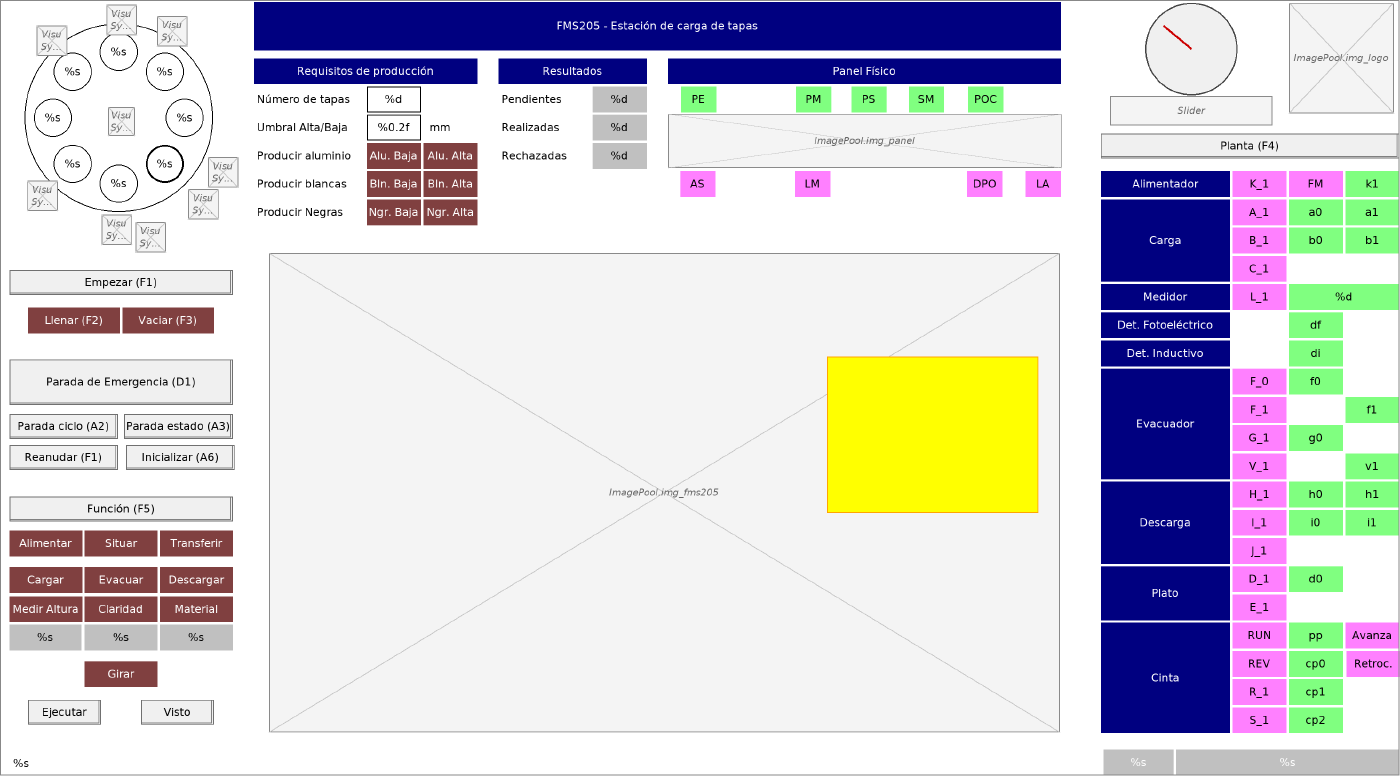
VISUALIZATION fms205visu  // 1488x825
    Rectangle (270,2 857x51), "FMS205 - Estación de carga de tapas", colour variable: MAIN.fbFMS205.dr.gmModeColor
        p3450524324: MAIN.fbFMS205.dr.gmModeColor
    Rectangle (270,62 237x27), "Requisitos de producción"
    Rectangle (530,62 157x27), "Resultados"
    Rectangle (710,62 417x27), "Panel Físico"
    Rectangle (270,92 157x27), "Número de tapas"
    Rectangle (390,92 57x27), "%d", text variable: MAIN.fbFMS205.ProdRequerida
    Rectangle (530,92 97x27), "Pendientes"
    Rectangle (630,92 57x27), "%d", text variable: MAIN.fbFMS205.ProdPendiente
    Rectangle (724,92 37x27), "PE", input disabled if: NOT MAIN.fbFMS205.dr.gmLocalHost
        toggle MAIN.fbFMS205.fbPanel.hwPE_Seta
    Rectangle (1029,92 37x27), "POC", input disabled if: NOT MAIN.fbFMS205.dr.gmLocalHost
        toggle MAIN.fbFMS205.fbPanel.hw.POC_PulsadorReset
    Rectangle (846,92 37x27), "PM", input disabled if: NOT MAIN.fbFMS205.dr.gmLocalHost
        toggle MAIN.fbFMS205.fbPanel.hw.PM_PulsadorMarcha
    Rectangle (966,92 37x27), "SM", input disabled if: NOT MAIN.fbFMS205.dr.gmLocalHost
        toggle MAIN.fbFMS205.fbPanel.hw.SM_SelecAutoManual
    Rectangle (270,122 117x27), "Umbral Alta/Baja"
    Rectangle (390,122 57x27), "%0.2f", text variable: MAIN.fbFMS205.fbPanel.cnUmbralAlta
        p4168582468: 'Atura en mm mínima para considerar que la tapa es alta'
    Rectangle (450,122 37x27), "mm"
    Rectangle (530,122 117x27), "Realizadas"
    Rectangle (630,122 57x27), "%d", text variable: MAIN.fbFMS205.ProdRealizada
    Rectangle (270,152 117x27), "Producir aluminio"
    Rectangle (390,152 57x27), "Alu. Baja"
        toggle MAIN.fbFMS205.fbPanel.cnProdAluBaja
    Rectangle (450,152 57x27), "Alu. Alta"
        toggle MAIN.fbFMS205.fbPanel.cnProdAluAlta
    Rectangle (530,152 117x27), "Rechazadas"
    Rectangle (630,152 57x27), "%d", text variable: MAIN.fbFMS205.ProdRechazada
    Button (1170,142 317x26), "Planta (F4)", tooltip "%s"
        p4168582468: MAIN.fbFMS205.fbPanel.ttF4_Planta
        toggle MAIN.fbFMS205.fbPanel.swF4_Planta
    Rectangle (270,182 117x27), "Producir blancas"
    Rectangle (390,182 57x27), "Bln. Baja"
        toggle MAIN.fbFMS205.fbPanel.cnProdBlaBaja
    Rectangle (450,182 57x27), "Bln. Alta"
        toggle MAIN.fbFMS205.fbPanel.cnProdBlaAlta
    Rectangle (1170,182 137x27), "Alimentador"
    Rectangle (1310,182 57x27), "K_1", input disabled if: NOT MAIN.fbFMS205.fbPanel.cnF4_Planta
        toggle MAIN.fbFMS205.mdAlimentador.K_1.uiValue p2164770859=TRUE
    Rectangle (1370,182 57x27), "FM", input disabled if: NOT MAIN.fbFMS205.fbPanel.cnF4_Planta
        toggle MAIN.fbFMS205.mdAlimentador.FM.uiValue
    Rectangle (1430,182 57x27), "k1", input disabled if: NOT MAIN.fbFMS205.fbPanel.cnF4_Planta
        toggle MAIN.fbFMS205.mdAlimentador.k1.uiValue
    Rectangle (723,182 37x27), "AS", input disabled if: NOT MAIN.fbFMS205.dr.gmLocalHost
        toggle MAIN.fbFMS205.fbPanel.hw.AS_AvisadorSonoro
    Rectangle (845,182 37x27), "LM", input disabled if: NOT MAIN.fbFMS205.dr.gmLocalHost
        toggle MAIN.fbFMS205.fbPanel.hw.LM_LamparaMarcha
    Rectangle (1028,182 37x27), "DPO", input disabled if: NOT MAIN.fbFMS205.dr.gmLocalHost
        toggle MAIN.fbFMS205.mdMedidorTapa.L_1.uiValue
    Rectangle (1090,182 37x27), "LA", input disabled if: NOT MAIN.fbFMS205.dr.gmLocalHost
        toggle MAIN.fbFMS205.fbPanel.hw.LA_LamparaAlarma
    Rectangle (270,212 117x27), "Producir Negras"
    Rectangle (390,212 57x27), "Ngr. Baja"
        toggle MAIN.fbFMS205.fbPanel.cnProdNegBaja
    Rectangle (450,212 57x27), "Ngr. Alta"
        toggle MAIN.fbFMS205.fbPanel.cnProdNegAlta
    Rectangle (1170,212 137x87), "Carga"
    Rectangle (1310,212 57x27), "A_1", input disabled if: NOT MAIN.fbFMS205.fbPanel.cnF4_Planta
        toggle MAIN.fbFMS205.mdPickAndPlaceCarga.HOR.uiValue
    Rectangle (1370,212 57x27), "a0", input disabled if: NOT MAIN.fbFMS205.fbPanel.cnF4_Planta
        toggle MAIN.fbFMS205.mdPickAndPlaceCarga.h0.uiValue
    Rectangle (1430,212 57x27), "a1", input disabled if: NOT MAIN.fbFMS205.fbPanel.cnF4_Planta
        toggle MAIN.fbFMS205.mdPickAndPlaceCarga.h1.uiValue
    Rectangle (1310,242 57x27), "B_1", input disabled if: NOT MAIN.fbFMS205.fbPanel.cnF4_Planta
        toggle MAIN.fbFMS205.mdPickAndPlaceCarga.VER.uiValue
    Rectangle (1370,242 57x27), "b0", input disabled if: NOT MAIN.fbFMS205.fbPanel.cnF4_Planta
        toggle MAIN.fbFMS205.mdPickAndPlaceCarga.v0.uiValue
    Rectangle (1430,242 57x27), "b1", input disabled if: NOT MAIN.fbFMS205.fbPanel.cnF4_Planta
        toggle MAIN.fbFMS205.mdPickAndPlaceCarga.v1.uiValue
    Rectangle (286,269 837x507), "Estacion"
    Button (10,287 237x26), "Empezar (F1)"
    Rectangle (30,327 97x27), "Llenar (F2)"
        toggle MAIN.fbFMS205.dr.fun_Llenar
    Rectangle (130,327 97x27), "Vaciar (F3)"
        toggle MAIN.fbFMS205.dr.fun_Vaciar
    Button (10,382 237x48), "Parada de Emergencia (D1)", tooltip "%s"
        p4168582468: MAIN.fbFMS205.fbPanel.ttPE_Seta
        toggle MAIN.fbFMS205.fbPanel.swPE_Seta
    Button (10,440 115x26), "Parada ciclo (A2)", input disabled if: not MAIN.fbFMS205.fbPanel.enA2_FinCiclo
        toggle MAIN.fbFMS205.fbPanel.swA2_FinCiclo
    Button (132,440 115x26), "Parada estado (A3)", input disabled if: not MAIN.fbFMS205.fbPanel.enA3_Estado
        toggle MAIN.fbFMS205.fbPanel.swA3_Estado
    Rectangle (1310,272 57x27), "C_1", input disabled if: NOT MAIN.fbFMS205.dr.bot_Planta
        toggle MAIN.fbFMS205.mdPickAndPlaceCarga.PIN.uiValue
    Rectangle (1170,302 137x27), "Medidor"
    Rectangle (1310,302 57x27), "L_1", input disabled if: NOT MAIN.fbFMS205.fbPanel.cnF4_Planta
        toggle MAIN.fbFMS205.mdMedidorTapa.L_1.uiValue
    Rectangle (1370,302 117x27), "%d", text variable: MAIN.fbFMS205.mdMedidorTapa.dh, input disabled if: NOT MAIN.fbFMS205.fbPanel.cnF4_Planta
    Rectangle (1170,332 137x27), "Det. Fotoeléctrico"
    Rectangle (1370,332 57x27), "df", input disabled if: NOT MAIN.fbFMS205.fbPanel.cnF4_Planta
        toggle MAIN.fbFMS205.mdDetectorFotoelectrico.df.uiValue
    Rectangle (1170,362 137x27), "Det. Inductivo"
    Rectangle (1370,362 57x27), "di", input disabled if: NOT MAIN.fbFMS205.fbPanel.cnF4_Planta
        toggle MAIN.fbFMS205.mdCaptadorInductivo.di.uiValue
    Rectangle (1170,392 137x117), "Evacuador"
    Rectangle (1310,392 57x27), "F_0", input disabled if: NOT MAIN.fbFMS205.fbPanel.cnF4_Planta
        toggle MAIN.fbFMS205.mdEvacuador.F_0.uiValue
    Rectangle (1370,392 57x27), "f0", input disabled if: NOT MAIN.fbFMS205.fbPanel.cnF4_Planta
        toggle MAIN.fbFMS205.mdEvacuador.f0.uiValue
    Button (10,528 237x26), "Función (F5)"
        toggle MAIN.fbFMS205.fbPanel.swF5_Funcion
    Rectangle (1310,422 57x27), "F_1", input disabled if: NOT MAIN.fbFMS205.fbPanel.cnF4_Planta
        toggle MAIN.fbFMS205.mdEvacuador.F_1.uiValue
    Rectangle (1430,422 57x27), "f1", input disabled if: NOT MAIN.fbFMS205.fbPanel.cnF4_Planta
        toggle MAIN.fbFMS205.mdEvacuador.f1.uiValue
    Rectangle (10,564 77x27), "Alimentar", input disabled if: not MAIN.fbFMS205.fbPanel.cnF5_Funcion
        toggle MAIN.fbFMS205.fbPanel.swF5_Alimentar
    Rectangle (90,703 77x27), "Girar", input disabled if: not MAIN.fbFMS205.fbPanel.cnF5_Funcion
        toggle MAIN.fbFMS205.fbPanel.swF5_Girar
    Rectangle (90,564 77x27), "Situar", input disabled if: not MAIN.fbFMS205.fbPanel.cnF5_Funcion
        toggle MAIN.fbFMS205.fbPanel.swF5_Situar
    Rectangle (10,634 77x27), "Medir Altura", input disabled if: not MAIN.fbFMS205.fbPanel.cnF5_Funcion
        toggle MAIN.fbFMS205.fbPanel.swF5_Medir
    Rectangle (90,634 77x27), "Claridad", input disabled if: not MAIN.fbFMS205.fbPanel.cnF5_Funcion
        toggle MAIN.fbFMS205.fbPanel.swF5_Claridad
    Rectangle (170,634 77x27), "Material", input disabled if: not MAIN.fbFMS205.fbPanel.cnF5_Funcion
        toggle MAIN.fbFMS205.fbPanel.swF5_Material
    Rectangle (10,664 76x27), "%s", text variable: MAIN.fbFMS205.mdMedidorTapa.strUi
    Rectangle (90,664 77x27), "%s", text variable: MAIN.fbFMS205.mdDetectorFotoelectrico.strUi
    Rectangle (170,664 77x27), "%s", text variable: MAIN.fbFMS205.mdCaptadorInductivo.strUi
    Rectangle (10,603 77x27), "Cargar", input disabled if: not MAIN.fbFMS205.fbPanel.cnF5_Funcion
        toggle MAIN.fbFMS205.fbPanel.swF5_Cargar
    Rectangle (90,603 77x27), "Evacuar", input disabled if: not MAIN.fbFMS205.fbPanel.cnF5_Funcion
        toggle MAIN.fbFMS205.fbPanel.swF5_Evacuar
    Rectangle (170,603 77x27), "Descargar", input disabled if: not MAIN.fbFMS205.fbPanel.cnF5_Funcion
        toggle MAIN.fbFMS205.fbPanel.swF5_Descargar
    Rectangle (170,564 77x27), "Transferir", input disabled if: not MAIN.fbFMS205.fbPanel.cnF5_Funcion
        toggle MAIN.fbFMS205.fbPanel.swF5_Transferir
    Button (30,744 77x26), "Ejecutar", input disabled if: not MAIN.fbFMS205.fbPanel.cnF5_Funcion
        tap MAIN.fbFMS205.fbPanel.swF5_Ejecutar
    Button (150,744 77x26), "Visto", input disabled if: not MAIN.fbFMS205.fbPanel.cnF5_Funcion
        tap MAIN.fbFMS205.fbPanel.swF5_Ack
    Rectangle (1310,452 57x27), "G_1", input disabled if: NOT MAIN.fbFMS205.fbPanel.cnF4_Planta
        toggle MAIN.fbFMS205.mdEvacuador.G_1.uiValue
    Rectangle (1370,452 57x27), "g0", input disabled if: NOT MAIN.fbFMS205.fbPanel.cnF4_Planta
        toggle MAIN.fbFMS205.mdEvacuador.g0.uiValue
    Rectangle (1310,482 57x27), "V_1", input disabled if: NOT MAIN.fbFMS205.fbPanel.cnF4_Planta
        toggle MAIN.fbFMS205.mdEvacuador.V_1.uiValue
    Rectangle (1430,482 57x27), "v1", input disabled if: NOT MAIN.fbFMS205.fbPanel.cnF4_Planta
        toggle MAIN.fbFMS205.mdEvacuador.v1.uiValue
    Rectangle (1170,512 137x87), "Descarga"
    Rectangle (1310,512 57x27), "H_1", input disabled if: NOT MAIN.fbFMS205.fbPanel.cnF4_Planta
        toggle MAIN.fbFMS205.mdPickAndPlaceDescarga.HOR.uiValue
    Rectangle (1370,512 57x27), "h0", input disabled if: NOT MAIN.fbFMS205.fbPanel.cnF4_Planta
        tap MAIN.fbFMS205.mdPickAndPlaceDescarga.h0.uiValue
        toggle MAIN.fbFMS205.mdPickAndPlaceDescarga.h0.uiValue
    Rectangle (1430,512 57x27), "h1", input disabled if: NOT MAIN.fbFMS205.fbPanel.cnF4_Planta
        toggle MAIN.fbFMS205.mdPickAndPlaceDescarga.h1.uiValue
    Rectangle (1310,542 57x27), "I_1", input disabled if: NOT MAIN.fbFMS205.fbPanel.cnF4_Planta
        toggle MAIN.fbFMS205.mdPickAndPlaceDescarga.VER.uiValue
    Rectangle (1370,542 57x27), "i0", input disabled if: NOT MAIN.fbFMS205.fbPanel.cnF4_Planta
        toggle MAIN.fbFMS205.mdPickAndPlaceDescarga.v0.uiValue
    Rectangle (1430,542 57x27), "i1", input disabled if: NOT MAIN.fbFMS205.fbPanel.cnF4_Planta
        toggle MAIN.fbFMS205.mdPickAndPlaceDescarga.v1.uiValue
    Rectangle (1310,572 57x27), "J_1", input disabled if: NOT MAIN.fbFMS205.fbPanel.cnF4_Planta
        toggle MAIN.fbFMS205.mdPickAndPlaceDescarga.PIN.uiValue
    Rectangle (1170,602 137x57), "Plato"
    Rectangle (1310,602 57x27), "D_1", input disabled if: NOT MAIN.fbFMS205.fbPanel.cnF4_Planta
        toggle MAIN.fbFMS205.mdPlatoDivisor.D_1.uiValue
    Rectangle (1370,602 57x27), "d0", input disabled if: NOT MAIN.fbFMS205.fbPanel.cnF4_Planta
        toggle MAIN.fbFMS205.mdPlatoDivisor.d0.uiValue
    Rectangle (1310,632 57x27), "E_1", input disabled if: NOT MAIN.fbFMS205.fbPanel.cnF4_Planta
        toggle MAIN.fbFMS205.mdPlatoDivisor.E_1.uiValue
    Rectangle (1170,662 137x117), "Cinta"
    Rectangle (1310,662 57x27), "RUN", input disabled if: NOT MAIN.fbFMS205.fbPanel.cnF4_Planta
        toggle MAIN.fbFMS205.mdCinta.RUN.uiValue
    Rectangle (1370,662 57x27), "pp", input disabled if: NOT MAIN.fbFMS205.fbPanel.cnF4_Planta
        toggle MAIN.fbFMS205.mdCinta.pp.uiValue
    Rectangle (1430,662 57x27), "Avanza", input disabled if: NOT MAIN.fbFMS205.fbPanel.cnF4_Planta
        toggle MAIN.fbFMS205.fbPanel.swF4_Avanza
    Rectangle (1310,692 57x27), "REV", input disabled if: NOT MAIN.fbFMS205.fbPanel.cnF4_Planta
        toggle MAIN.fbFMS205.mdCinta.REV.uiValue
    Rectangle (1370,692 57x27), "cp0", input disabled if: NOT MAIN.fbFMS205.fbPanel.cnF4_Planta
        toggle MAIN.fbFMS205.mdCinta.cp0.uiValue
    Rectangle (1431,692 57x27), "Retroc.", input disabled if: NOT MAIN.fbFMS205.fbPanel.cnF4_Planta
        toggle MAIN.fbFMS205.fbPanel.swF4_Retroc
    Rectangle (1310,722 57x27), "R_1", input disabled if: NOT MAIN.fbFMS205.fbPanel.cnF4_Planta
        toggle MAIN.fbFMS205.mdCinta.R_1.uiValue
    Rectangle (1370,722 57x27), "cp1", input disabled if: NOT MAIN.fbFMS205.fbPanel.cnF4_Planta
        toggle MAIN.fbFMS205.mdCinta.cp1.uiValue
    Rectangle (1310,752 57x27), "S_1", input disabled if: NOT MAIN.fbFMS205.fbPanel.cnF4_Planta
        toggle MAIN.fbFMS205.mdCinta.S_1.uiValue
    Rectangle (1370,752 57x27), "cp2", input disabled if: NOT MAIN.fbFMS205.fbPanel.cnF4_Planta
        toggle MAIN.fbFMS205.mdCinta.cp2.uiValue
    Rectangle (11,798 1117x27), "%s", text variable: main.fbFMS205.fbPanel.swMensaje
    Rectangle (1173,797 74x27), "%s", text variable: MAIN.fbFMS205.dr.gmModeName, colour variable: MAIN.fbFMS205.dr.gmModeColor
        p3450524324: MAIN.fbFMS205.dr.gmModeColor
    Rectangle (1250,797 237x27), "%s", text variable: MAIN.fbFMS205.dr.gmModeDescr, colour variable: MAIN.fbFMS205.dr.gmModeColor
        p3450524324: MAIN.fbFMS205.dr.gmModeColor
    Ellipse (26,25 200x200)
    Ellipse (176,105 40x40), "%s", text variable: MAIN.fbFMS205.sectores[7].strUi, colour variable: MAIN.fbFMS205.sectores[7].ColorSector
        p2277200375: MAIN.fbFMS205.angulo+MAIN.fbFMS205.anguloanim
    Ellipse (155,154 40x40), "%s", text variable: MAIN.fbFMS205.sectores[0].strUi, colour variable: MAIN.fbFMS205.sectores[0].ColorSector
        p2277200375: MAIN.fbFMS205.angulo+MAIN.fbFMS205.anguloanim
    Ellipse (106,175 40x40), "%s", text variable: MAIN.fbFMS205.sectores[1].strUi, colour variable: MAIN.fbFMS205.sectores[1].ColorSector
        p2277200375: MAIN.fbFMS205.angulo+MAIN.fbFMS205.anguloanim
    Ellipse (57,154 40x40), "%s", text variable: MAIN.fbFMS205.sectores[2].strUi, colour variable: MAIN.fbFMS205.sectores[2].ColorSector
        p2277200375: MAIN.fbFMS205.angulo+MAIN.fbFMS205.anguloanim
    Ellipse (36,105 40x40), "%s", text variable: MAIN.fbFMS205.sectores[3].strUi, colour variable: MAIN.fbFMS205.sectores[3].ColorSector
        p2277200375: MAIN.fbFMS205.angulo+MAIN.fbFMS205.anguloanim
    Ellipse (57,56 40x40), "%s", text variable: MAIN.fbFMS205.sectores[4].strUi, colour variable: MAIN.fbFMS205.sectores[4].ColorSector
        p2277200375: MAIN.fbFMS205.angulo+MAIN.fbFMS205.anguloanim
    Ellipse (106,35 40x40), "%s", text variable: MAIN.fbFMS205.sectores[5].strUi, colour variable: MAIN.fbFMS205.sectores[5].ColorSector
        p2277200375: MAIN.fbFMS205.angulo+MAIN.fbFMS205.anguloanim
    Ellipse (155,56 40x40), "%s", text variable: MAIN.fbFMS205.sectores[6].strUi, colour variable: MAIN.fbFMS205.sectores[6].ColorSector
        p2277200375: MAIN.fbFMS205.angulo+MAIN.fbFMS205.anguloanim
    Image (286,269 840x509), image: ImagePool.img_fms205
    Image (1370,3 111x117), image: ImagePool.img_logo
    Image (710,121 418x57), image: ImagePool.img_panel
    Rectangle (905,92 37x27), "PS", input disabled if: NOT MAIN.fbFMS205.dr.gmLocalHost
        toggle MAIN.fbFMS205.fbPanel.hw.PS_PulsadorStop
    Image (115,114 28x30), invisible if: MAIN.fbFMS205.mdPlatoDivisor.Ready, image: VisuSymbols.Symbols.ArrowHalfLeftUp
    Image (221,167 32x32), invisible if: MAIN.fbFMS205.mdAlimentador.Ready, image: VisuSymbols.Symbols.ArrowBoldDown
    Image (167,17 32x32), invisible if: not MAIN.fbFMS205.mdMedidorTapa.IsActive, image: VisuSymbols.Symbols.ArrowBoldDown
    Image (113,5 32x32), invisible if: MAIN.fbFMS205.mdDetectorFotoelectrico.Ready, image: VisuSymbols.Symbols.Download
    Image (39,27 32x32), invisible if: MAIN.fbFMS205.mdCaptadorInductivo.Ready, image: VisuSymbols.Symbols.Download
    Image (29,192 32x32), invisible if: MAIN.fbFMS205.mdEvacuador.Ready, image: VisuSymbols.Symbols.ArrowBoldLeftDown
    Image (108,228 32x32), invisible if: MAIN.fbFMS205.mdPickAndPlaceDescarga.Ready, image: VisuSymbols.Symbols.ArrowBoldDown
    Image (144,236 32x32), invisible if: MAIN.fbFMS205.mdCinta.Ready, image: VisuSymbols.Symbols.ArrowBoldRight
    Image (200,201 32x32), invisible if: MAIN.fbFMS205.mdPickAndPlaceCarga.Ready, image: VisuSymbols.Symbols.ArrowBoldLeftUp
    Meter180 (1171,3 190x98), value: MAIN.fbFMS205.dr.Speed, style: Meter-Meter180-Gray, scale format: %.1f, scale 0..200
    Slider (1180,102 172x31), variable: MAIN.fbFMS205.dr.Speed, scale 1..200
    Rectangle (879,379 224x166), invisible if: NOT MAIN.fbFMS205.mdPickAndPlaceCarga.IsActive
        p2738717112: MAIN.fbFMS205.mdPickAndPlaceCarga.VER.uiUp
    Button (10,473 115x26), "Reanudar (F1)", input disabled if: not MAIN.fbFMS205.fbPanel.enF1_Reanduar
        tap MAIN.fbFMS205.fbPanel.swF1_Reanudar
    Button (134,473 115x26), "Inicializar (A6)"
        tap MAIN.fbFMS205.fbPanel.swA6_Inicializar
END_VISUALIZATION

(* stored: Version 1.1.0.1, ProductVersion 3.1.4024.11
   Visu fms205visu: Id {024cfbd6-56e0-4061-82c5-347b4091fefa} *)
